TYPE STATE:
    STRUCT
        curTime: LREAL;
        dvar_M_aut_x AT %Q*: DINT;
        dvar_M_aut_y AT %Q*: DINT;
        dvar_M_aut_z AT %Q*: DINT;
    END_STRUCT
END_TYPE

(* stored: ProductVersion 3.1.0.18, Version 1.1.0.1 *)
